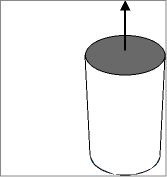
VISUALIZATION VISU_Tube_Top_8  // 167x177
VAR_IN_OUT
	azi : LREAL;
END_VAR
    Ellipse (90,135 70x40)
        p2858320360: azi
    Polygon (85,55) (165,55) (160,155) (156,163) (151,168) (144,171) (134,174) (124,174) (114,174) (107,171) (102,169) (95,164) (90,155)
        p2858320360: azi
    Ellipse (85,35 80x40)
        p2858320360: azi
    Polygon (120,10) (125,0) (130,10)
        p2858320360: azi
    Polyline (125,50) (125,10)
        p2858320360: azi
    Polyline (160,155) (165,55)
        p2858320360: azi
    Polyline (90,155) (85,55)
        p2858320360: azi
END_VISUALIZATION

(* stored: Version 1.1.0.1, ProductVersion 3.1.4019.2
   Visu VISU_Tube_Top_8: Id {af7d9f94-2a48-4574-8bbe-4d26d4d0fb9c} *)
